(* IEC 61131-3 sources: PLC_MixingTank/MixingTank/FB, 4 files *)

(* ---- FB_PID_Var.st ---- *)
FUNCTION_BLOCK FB_PID
VAR_INPUT
    SetPoint : REAL;
    ProcessValue : REAL;
    Kp : REAL;
    Ti : REAL;
    Td : REAL;
    CycleTime : REAL;
    Enable : BOOL;
    OutMin : REAL := 0.0;
    OutMax : REAL := 100.0;
END_VAR

VAR_OUTPUT
    Out : REAL;
    Error : REAL;
END_VAR

VAR
    PrevError : REAL;
    Integral : REAL;
    Derivative : REAL;
    RawOut : REAL;
END_VAR

(* ---- FB_TankLevelSim_Var.st ---- *)
FUNCTION_BLOCK FB_TankLevelSim
VAR_INPUT
    OilPumpActive : BOOL;
    IngredientTrigger : BOOL;
    DrainValveActive : BOOL;

    Execute : BOOL;
    Reset : BOOL;

    OilFillRate : REAL := 5.0;
    IngredientAmount : REAL := 50.0;
    DrainRate : REAL := 8.0;
END_VAR

VAR_OUTPUT
    SimulatedLevel : REAL := 0.0;
END_VAR

VAR
    RawTrig : R_TRIG;
    dLevel : REAL;
END_VAR

(* ---- FB_TankLevelSim_Exe.st ---- *)
RawTrig(CLK := IngredientTrigger);

IF Reset THEN
    SimulatedLevel := 0.0;
ELSE
    IF RawTrig.Q THEN
        SimulatedLevel := SimulatedLevel + IngredientAmount;
    END_IF

    IF Execute THEN
        dLevel := 0.0;

        IF OilPumpActive THEN
            dLevel := dLevel + OilFillRate;
        END_IF

        IF DrainValveActive THEN
            dLevel := dLevel - DrainRate;
        END_IF

        SimulatedLevel := SimulatedLevel + dLevel;
    END_IF

    IF SimulatedLevel < 0.0 THEN
        SimulatedLevel := 0.0;
    END_IF
END_IF

(* ---- FB_TankTempSim_Exe.st ---- *)
IF Reset THEN
    SimulatedTemp := AmbientTemp;
ELSIF Execute THEN
    dTemp := (SteamValveInput / 100.0) * MaxHeatingPerSec - HeatLostCoeff * (SimulatedTemp - AmbientTemp);
    SimulatedTemp := SimulatedTemp + dTemp;
END_IF
